FUNCTION_BLOCK FB_TransferirPale_SFC

VAR_INPUT
    // SFC-Flags
    SFCPause: BOOL;
    SFCReset: BOOL;
    
    // Sincronizacion
    Benido: BOOL := TRUE;
    Ejecuta: BOOL;
    
    // Parametros de tiempo
    TpoCintaRetenedor: TIME := T#1S;
    TpoPaleSalida: TIME := T#1S;
    TpoPaleTransferencia: TIME := T#1S;

    PresenciaPale AT %I* : BOOL;
END_VAR
VAR_OUTPUT
   
    // Sincronizacion    
    Acabhe: BOOL;
    ListoKalisto: BOOL;
    
    CintaActiva AT %Q* : BOOL;
    RetenedorBaja AT %Q* : BOOL;
END_VAR
VAR  
END_VAR

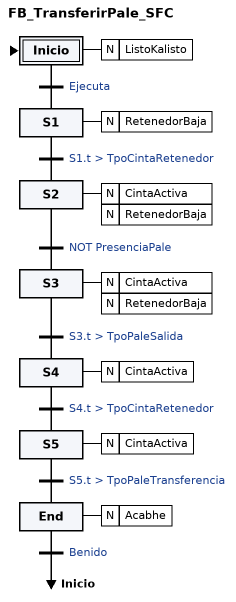
INITIAL_STEP Inicio:
    ListoKalisto(N);
END_STEP
TRANSITION FROM Inicio TO S1
    := Ejecuta;
END_TRANSITION
STEP S1:
    RetenedorBaja(N);
END_STEP
TRANSITION FROM S1 TO S2
    := S1.t > TpoCintaRetenedor;
END_TRANSITION
STEP S2:
    CintaActiva(N);
    RetenedorBaja(N);
END_STEP
TRANSITION FROM S2 TO S3
    := NOT PresenciaPale;
END_TRANSITION
STEP S3:
    CintaActiva(N);
    RetenedorBaja(N);
END_STEP
TRANSITION FROM S3 TO S4
    := S3.t > TpoPaleSalida;
END_TRANSITION
STEP S4:
    CintaActiva(N);
END_STEP
TRANSITION FROM S4 TO S5
    := S4.t > TpoCintaRetenedor;
END_TRANSITION
STEP S5:
    CintaActiva(N);
END_STEP
TRANSITION FROM S5 TO End
    := S5.t > TpoPaleTransferencia;
END_TRANSITION
STEP End:
    Acabhe(N);
END_STEP
TRANSITION FROM End TO Inicio
    := Benido;
END_TRANSITION

END_FUNCTION_BLOCK

(* stored: Version 1.1.0.1, ProductVersion 3.1.4024.12
   POU FB_TransferirPale_SFC: Id {4d60dea1-7dc4-49b2-8ad0-0eb99b5fb071}, SpecialFunc None *)
